   1:L PR[91] R[100]mm/sec CNT100;
   1:  PR[91,1] = PR[90,1] + 37.532;
   1:  PR[91,2] = PR[90,2] + 2.795;
   1:L PR[91] R[100]mm/sec CNT100;
   1:  PR[91,1] = PR[90,1] + 37.500;
   1:  PR[91,2] = PR[90,2] + 3.023;
   1:L PR[91] R[100]mm/sec CNT100;
   1:  PR[91,1] = PR[90,1] + 36.763;
   1:  PR[91,2] = PR[90,2] + 5.831;
   1:L PR[91] R[100]mm/sec CNT100;
   1:  PR[91,1] = PR[90,1] + 35.316;
   1:  PR[91,2] = PR[90,2] + 9.032;
   1:L PR[91] R[100]mm/sec CNT100;
   1:  PR[91,1] = PR[90,1] + 33.687;
   1:  PR[91,2] = PR[90,2] + 11.493;
   1:L PR[91] R[100]mm/sec CNT100;
   1:  PR[91,1] = PR[90,1] + 33.253;
   1:  PR[91,2] = PR[90,2] + 12.032;
   1:L PR[91] R[100]mm/sec CNT100;
   1:  PR[91,1] = PR[90,1] + 31.314;
   1:  PR[91,2] = PR[90,2] + 14.124;
   1:L PR[91] R[100]mm/sec CNT100;
   1:  PR[91,1] = PR[90,1] + 29.228;
   1:  PR[91,2] = PR[90,2] + 15.750;
   1:L PR[91] R[100]mm/sec CNT100;
   1:  PR[91,1] = PR[90,1] + 28.265;
   1:  PR[91,2] = PR[90,2] + 16.449;
   1:L PR[91] R[100]mm/sec CNT100;
   1:  PR[91,1] = PR[90,1] + 26.032;
   1:  PR[91,2] = PR[90,2] + 17.693;
   1:L PR[91] R[100]mm/sec CNT100;
   1:  PR[91,1] = PR[90,1] + 23.783;
   1:  PR[91,2] = PR[90,2] + 18.520;
   1:L PR[91] R[100]mm/sec CNT100;
   1:  PR[91,1] = PR[90,1] + 22.146;
   1:  PR[91,2] = PR[90,2] + 19.160;
   1:L PR[91] R[100]mm/sec CNT100;
   1:  PR[91,1] = PR[90,1] + 19.988;
   1:  PR[91,2] = PR[90,2] + 19.606;
   1:L PR[91] R[100]mm/sec CNT100;
   1:  PR[91,1] = PR[90,1] + 17.828;
   1:  PR[91,2] = PR[90,2] + 19.862;
   1:L PR[91] R[100]mm/sec CNT100;
   1:  PR[91,1] = PR[90,1] + 15.729;
   1:  PR[91,2] = PR[90,2] + 19.971;
   1:L PR[91] R[100]mm/sec CNT100;
   1:  PR[91,1] = PR[90,1] + 13.857;
   1:  PR[91,2] = PR[90,2] + 19.781;
   1:L PR[91] R[100]mm/sec CNT100;
   1:  PR[91,1] = PR[90,1] + 11.168;
   1:  PR[91,2] = PR[90,2] + 19.409;
   1:L PR[91] R[100]mm/sec CNT100;
   1:  PR[91,1] = PR[90,1] + 9.530;
   1:  PR[91,2] = PR[90,2] + 18.985;
   1:L PR[91] R[100]mm/sec CNT100;
   1:  PR[91,1] = PR[90,1] + 8.064;
   1:  PR[91,2] = PR[90,2] + 18.343;
   1:L PR[91] R[100]mm/sec CNT100;
   1:  PR[91,1] = PR[90,1] + 5.139;
   1:  PR[91,2] = PR[90,2] + 17.121;
   1:L PR[91] R[100]mm/sec CNT100;
   1:  PR[91,1] = PR[90,1] + 3.965;
   1:  PR[91,2] = PR[90,2] + 16.371;
   1:L PR[91] R[100]mm/sec CNT100;
   1:  PR[91,1] = PR[90,1] + 3.405;
   1:  PR[91,2] = PR[90,2] + 15.985;
   1:L PR[91] R[100]mm/sec CNT100;
   1:  PR[91,1] = PR[90,1] + 2.387;
   1:  PR[91,2] = PR[90,2] + 15.179;
   1:L PR[91] R[100]mm/sec CNT100;
   1:  PR[91,1] = PR[90,1] + 2.008;
   1:  PR[91,2] = PR[90,2] + 14.843;
   1:L PR[91] R[100]mm/sec CNT100;
   1:  PR[91,1] = PR[90,1] + 1.924;
   1:  PR[91,2] = PR[90,2] + 14.787;
   1:L PR[91] R[100]mm/sec CNT100;
   1:  PR[91,1] = PR[90,1] + 1.541;
   1:  PR[91,2] = PR[90,2] + 14.416;
   1:L PR[91] R[100]mm/sec CNT100;
   1:  PR[91,1] = PR[90,1] + 0.779;
   1:  PR[91,2] = PR[90,2] + 14.285;
   1:L PR[91] R[100]mm/sec CNT100;
   1:  PR[91,1] = PR[90,1] + 0.419;
   1:  PR[91,2] = PR[90,2] + 14.088;
   1:L PR[91] R[100]mm/sec CNT100;
   1:  PR[91,1] = PR[90,1] + -0.391;
   1:L PR[91] R[100]mm/sec CNT100;
   1:  PR[91] = PR[90];
   1:  PR[91,1] = PR[90,1] + -1.750;
   1:  PR[91,2] = PR[90,2] + 15.019;
   1:  PR[91,3] = PR[90,3] + 33.245;
   1:L PR[91] R[100]mm/sec CNT100;
   1:  PR[91,1] = PR[90,1] + -1.966;
   1:  PR[91,2] = PR[90,2] + 15.226;
   1:L PR[91] R[100]mm/sec CNT100;
   1:  PR[91,1] = PR[90,1] + -3.004;
   1:  PR[91,2] = PR[90,2] + 16.046;
   1:L PR[91] R[100]mm/sec CNT100;
   1:  PR[91,1] = PR[90,1] + -3.762;
   1:  PR[91,2] = PR[90,2] + 16.531;
   1:L PR[91] R[100]mm/sec CNT100;
   1:  PR[91,1] = PR[90,1] + -4.723;
   1:  PR[91,2] = PR[90,2] + 17.176;
   1:L PR[91] R[100]mm/sec CNT100;
   1:  PR[91,1] = PR[90,1] + -6.056;
   1:  PR[91,2] = PR[90,2] + 17.758;
   1:L PR[91] R[100]mm/sec CNT100;
   1:  PR[91,1] = PR[90,1] + -9.172;
   1:  PR[91,2] = PR[90,2] + 19.064;
   1:L PR[91] R[100]mm/sec CNT100;
   1:  PR[91,1] = PR[90,1] + -10.666;
   1:  PR[91,2] = PR[90,2] + 19.451;
   1:L PR[91] R[100]mm/sec CNT100;
   1:  PR[91,1] = PR[90,1] + -12.540;
   1:  PR[91,2] = PR[90,2] + 19.646;
   1:L PR[91] R[100]mm/sec CNT100;
   1:  PR[91,1] = PR[90,1] + -15.381;
   1:  PR[91,2] = PR[90,2] + 20.034;
   1:L PR[91] R[100]mm/sec CNT100;
   1:  PR[91,1] = PR[90,1] + -17.322;
   1:  PR[91,2] = PR[90,2] + 19.931;
   1:L PR[91] R[100]mm/sec CNT100;
   1:  PR[91,1] = PR[90,1] + -19.724;
   1:  PR[91,2] = PR[90,2] + 19.647;
   1:L PR[91] R[100]mm/sec CNT100;
   1:  PR[91,1] = PR[90,1] + -21.764;
   1:  PR[91,2] = PR[90,2] + 19.224;
   1:L PR[91] R[100]mm/sec CNT100;
   1:  PR[91,1] = PR[90,1] + -24.013;
   1:  PR[91,2] = PR[90,2] + 18.389;
   1:L PR[91] R[100]mm/sec CNT100;
   1:  PR[91,1] = PR[90,1] + -25.716;
   1:  PR[91,2] = PR[90,2] + 17.723;
   1:L PR[91] R[100]mm/sec CNT100;
   1:  PR[91,1] = PR[90,1] + -27.825;
   1:  PR[91,2] = PR[90,2] + 16.541;
   1:L PR[91] R[100]mm/sec CNT100;
   1:  PR[91,1] = PR[90,1] + -30.010;
   1:  PR[91,2] = PR[90,2] + 14.841;
   1:L PR[91] R[100]mm/sec CNT100;
   1:  PR[91,1] = PR[90,1] + -31.019;
   1:  PR[91,2] = PR[90,2] + 14.106;
   1:L PR[91] R[100]mm/sec CNT100;
   1:  PR[91,1] = PR[90,1] + -32.838;
   1:  PR[91,2] = PR[90,2] + 12.142;
   1:L PR[91] R[100]mm/sec CNT100;
   1:  PR[91,1] = PR[90,1] + -33.428;
   1:  PR[91,2] = PR[90,2] + 11.409;
   1:L PR[91] R[100]mm/sec CNT100;
   1:  PR[91,1] = PR[90,1] + -34.956;
   1:  PR[91,2] = PR[90,2] + 9.087;
   1:L PR[91] R[100]mm/sec CNT100;
   1:  PR[91,1] = PR[90,1] + -36.446;
   1:  PR[91,2] = PR[90,2] + 5.748;
   1:L PR[91] R[100]mm/sec CNT100;
   1:  PR[91,1] = PR[90,1] + -37.137;
   1:  PR[91,2] = PR[90,2] + 3.081;
   1:L PR[91] R[100]mm/sec CNT100;
   1:  PR[91,1] = PR[90,1] + -37.374;
   1:  PR[91,2] = PR[90,2] + 0.115;
   1:L PR[91] R[100]mm/sec CNT100;
   1:  PR[91,1] = PR[90,1] + -37.439;
   1:  PR[91,2] = PR[90,2] + -0.354;
   1:L PR[91] R[100]mm/sec CNT100;
   1:  PR[91,1] = PR[90,1] + -37.214;
   1:  PR[91,2] = PR[90,2] + -3.186;
   1:L PR[91] R[100]mm/sec CNT100;
   1:  PR[91,1] = PR[90,1] + -37.147;
   1:  PR[91,2] = PR[90,2] + -3.665;
   1:L PR[91] R[100]mm/sec CNT100;
   1:  PR[91,1] = PR[90,1] + -36.446;
   1:  PR[91,2] = PR[90,2] + -6.371;
   1:L PR[91] R[100]mm/sec CNT100;
   1:  PR[91,1] = PR[90,1] + -35.239;
   1:  PR[91,2] = PR[90,2] + -9.063;
   1:L PR[91] R[100]mm/sec CNT100;
   1:  PR[91,1] = PR[90,1] + -34.952;
   1:  PR[91,2] = PR[90,2] + -9.717;
   1:L PR[91] R[100]mm/sec CNT100;
   1:  PR[91,1] = PR[90,1] + -33.427;
   1:  PR[91,2] = PR[90,2] + -12.034;
   1:L PR[91] R[100]mm/sec CNT100;
   1:  PR[91,1] = PR[90,1] + -32.835;
   1:  PR[91,2] = PR[90,2] + -12.768;
   1:L PR[91] R[100]mm/sec CNT100;
   1:  PR[91,1] = PR[90,1] + -30.998;
   1:  PR[91,2] = PR[90,2] + -14.752;
   1:L PR[91] R[100]mm/sec CNT100;
   1:  PR[91,1] = PR[90,1] + -29.002;
   1:  PR[91,2] = PR[90,2] + -16.314;
   1:L PR[91] R[100]mm/sec CNT100;
   1:  PR[91,1] = PR[90,1] + -27.839;
   1:  PR[91,2] = PR[90,2] + -17.157;
   1:L PR[91] R[100]mm/sec CNT100;
   1:  PR[91,1] = PR[90,1] + -25.720;
   1:  PR[91,2] = PR[90,2] + -18.345;
   1:L PR[91] R[100]mm/sec CNT100;
   1:  PR[91,1] = PR[90,1] + -23.597;
   1:  PR[91,2] = PR[90,2] + -19.129;
   1:L PR[91] R[100]mm/sec CNT100;
   1:  PR[91,1] = PR[90,1] + -21.738;
   1:  PR[91,2] = PR[90,2] + -19.854;
   1:L PR[91] R[100]mm/sec CNT100;
   1:  PR[91,1] = PR[90,1] + -19.710;
   1:  PR[91,2] = PR[90,2] + -20.274;
   1:L PR[91] R[100]mm/sec CNT100;
   1:  PR[91,1] = PR[90,1] + -17.303;
   1:  PR[91,2] = PR[90,2] + -20.555;
   1:L PR[91] R[100]mm/sec CNT100;
   1:  PR[91,1] = PR[90,1] + -15.334;
   1:  PR[91,2] = PR[90,2] + -20.659;
   1:L PR[91] R[100]mm/sec CNT100;
   1:  PR[91,1] = PR[90,1] + -13.585;
   1:  PR[91,2] = PR[90,2] + -20.483;
   1:L PR[91] R[100]mm/sec CNT100;
   1:  PR[91,1] = PR[90,1] + -10.663;
   1:  PR[91,2] = PR[90,2] + -20.074;
   1:L PR[91] R[100]mm/sec CNT100;
   1:  PR[91,1] = PR[90,1] + -9.156;
   1:  PR[91,2] = PR[90,2] + -19.684;
   1:L PR[91] R[100]mm/sec CNT100;
   1:  PR[91,1] = PR[90,1] + -7.803;
   1:  PR[91,2] = PR[90,2] + -19.090;
   1:L PR[91] R[100]mm/sec CNT100;
   1:  PR[91,1] = PR[90,1] + -4.609;
   1:  PR[91,2] = PR[90,2] + -17.729;
   1:L PR[91] R[100]mm/sec CNT100;
   1:  PR[91,1] = PR[90,1] + -3.572;
   1:  PR[91,2] = PR[90,2] + -17.067;
   1:L PR[91] R[100]mm/sec CNT100;
   1:  PR[91,1] = PR[90,1] + -2.643;
   1:  PR[91,2] = PR[90,2] + -16.396;
   1:L PR[91] R[100]mm/sec CNT100;
   1:  PR[91,1] = PR[90,1] + -1.685;
   1:  PR[91,2] = PR[90,2] + -15.558;
   1:L PR[91] R[100]mm/sec CNT100;
   1:  PR[91,1] = PR[90,1] + -0.884;
   1:  PR[91,2] = PR[90,2] + -15.285;
   1:L PR[91] R[100]mm/sec CNT100;
   1:  PR[91,1] = PR[90,1] + -0.313;
   1:  PR[91,2] = PR[90,2] + -14.848;
   1:L PR[91] R[100]mm/sec CNT100;
   1:  PR[91,1] = PR[90,1] + 0.513;
   1:  PR[91,2] = PR[90,2] + -15.142;
   1:L PR[91] R[100]mm/sec CNT100;
   1:  PR[91,1] = PR[90,1] + 1.632;
   1:  PR[91,2] = PR[90,2] + -15.342;
   1:L PR[91] R[100]mm/sec CNT100;
   1:  PR[91,1] = PR[90,1] + 1.864;
   1:  PR[91,2] = PR[90,2] + -15.606;
   1:L PR[91] R[100]mm/sec CNT100;
   1:  PR[91,1] = PR[90,1] + 1.960;
   1:  PR[91,2] = PR[90,2] + -15.664;
   1:L PR[91] R[100]mm/sec CNT100;
   1:  PR[91,1] = PR[90,1] + 2.771;
   1:  PR[91,2] = PR[90,2] + -16.374;
   1:L PR[91] R[100]mm/sec CNT100;
   1:  PR[91,1] = PR[90,1] + 3.240;
   1:  PR[91,2] = PR[90,2] + -16.675;
   1:L PR[91] R[100]mm/sec CNT100;
   1:  PR[91,1] = PR[90,1] + 3.869;
   1:  PR[91,2] = PR[90,2] + -17.123;
   1:L PR[91] R[100]mm/sec CNT100;
   1:  PR[91,1] = PR[90,1] + 4.780;
   1:  PR[91,2] = PR[90,2] + -17.738;
   1:L PR[91] R[100]mm/sec CNT100;
   1:  PR[91,1] = PR[90,1] + 9.302;
   1:  PR[91,2] = PR[90,2] + -19.679;
   1:L PR[91] R[100]mm/sec CNT100;
   1:  PR[91,1] = PR[90,1] + 10.793;
   1:  PR[91,2] = PR[90,2] + -20.065;
   1:L PR[91] R[100]mm/sec CNT100;
   1:  PR[91,1] = PR[90,1] + 12.664;
   1:  PR[91,2] = PR[90,2] + -20.262;
   1:L PR[91] R[100]mm/sec CNT100;
   1:  PR[91,1] = PR[90,1] + 15.511;
   1:  PR[91,2] = PR[90,2] + -20.658;
   1:L PR[91] R[100]mm/sec CNT100;
   1:  PR[91,1] = PR[90,1] + 17.443;
   1:  PR[91,2] = PR[90,2] + -20.557;
   1:L PR[91] R[100]mm/sec CNT100;
   1:  PR[91,1] = PR[90,1] + 19.851;
   1:  PR[91,2] = PR[90,2] + -20.277;
   1:L PR[91] R[100]mm/sec CNT100;
   1:  PR[91,1] = PR[90,1] + 21.888;
   1:  PR[91,2] = PR[90,2] + -19.855;
   1:L PR[91] R[100]mm/sec CNT100;
   1:  PR[91,1] = PR[90,1] + 24.142;
   1:  PR[91,2] = PR[90,2] + -19.022;
   1:L PR[91] R[100]mm/sec CNT100;
   1:  PR[91,1] = PR[90,1] + 25.852;
   1:  PR[91,2] = PR[90,2] + -18.358;
   1:L PR[91] R[100]mm/sec CNT100;
   1:  PR[91,1] = PR[90,1] + 27.952;
   1:  PR[91,2] = PR[90,2] + -17.187;
   1:L PR[91] R[100]mm/sec CNT100;
   1:  PR[91,1] = PR[90,1] + 30.119;
   1:  PR[91,2] = PR[90,2] + -15.508;
   1:L PR[91] R[100]mm/sec CNT100;
   1:  PR[91,1] = PR[90,1] + 31.133;
   1:  PR[91,2] = PR[90,2] + -14.771;
   1:L PR[91] R[100]mm/sec CNT100;
   1:  PR[91,1] = PR[90,1] + 32.956;
   1:  PR[91,2] = PR[90,2] + -12.805;
   1:L PR[91] R[100]mm/sec CNT100;
   1:  PR[91,1] = PR[90,1] + 33.551;
   1:  PR[91,2] = PR[90,2] + -12.066;
   1:L PR[91] R[100]mm/sec CNT100;
   1:  PR[91,1] = PR[90,1] + 35.101;
   1:  PR[91,2] = PR[90,2] + -9.725;
   1:L PR[91] R[100]mm/sec CNT100;
   1:  PR[91,1] = PR[90,1] + 36.351;
   1:  PR[91,2] = PR[90,2] + -6.972;
   1:L PR[91] R[100]mm/sec CNT100;
   1:  PR[91,1] = PR[90,1] + 36.587;
   1:  PR[91,2] = PR[90,2] + -6.435;
   1:L PR[91] R[100]mm/sec CNT100;
   1:  PR[91,1] = PR[90,1] + 37.280;
   1:  PR[91,2] = PR[90,2] + -3.795;
   1:L PR[91] R[100]mm/sec CNT100;
   1:  PR[91,1] = PR[90,1] + 37.531;
   1:  PR[91,2] = PR[90,2] + -0.740;
   1:L PR[91] R[100]mm/sec CNT100;
   1:  PR[91,1] = PR[90,1] + 37.596;
   1:  PR[91,2] = PR[90,2] + -0.271;
   1:L PR[91] R[100]mm/sec CNT100;
   1:  PR[91,1] = PR[90,1] + 37.358;
   1:  PR[91,2] = PR[90,2] + 2.651;
   1:L PR[91] R[100]mm/sec CNT100;
   1:  PR[91,1] = PR[90,1] + 37.291;
   1:  PR[91,2] = PR[90,2] + 3.131;
   1:L PR[91] R[100]mm/sec CNT100;
   1:  PR[91,1] = PR[90,1] + 36.589;
   1:  PR[91,2] = PR[90,2] + 5.804;
   1:L PR[91] R[100]mm/sec CNT100;
   1:  PR[91,1] = PR[90,1] + 35.101;
   1:  PR[91,2] = PR[90,2] + 9.100;
   1:L PR[91] R[100]mm/sec CNT100;
   1:  PR[91,1] = PR[90,1] + 33.552;
   1:  PR[91,2] = PR[90,2] + 11.440;
   1:L PR[91] R[100]mm/sec CNT100;
   1:  PR[91,1] = PR[90,1] + 32.959;
   1:  PR[91,2] = PR[90,2] + 12.178;
   1:L PR[91] R[100]mm/sec CNT100;
   1:  PR[91,1] = PR[90,1] + 31.120;
   1:  PR[91,2] = PR[90,2] + 14.162;
   1:L PR[91] R[100]mm/sec CNT100;
   1:  PR[91,1] = PR[90,1] + 29.140;
   1:  PR[91,2] = PR[90,2] + 15.704;
   1:L PR[91] R[100]mm/sec CNT100;
   1:  PR[91,1] = PR[90,1] + 27.979;
   1:  PR[91,2] = PR[90,2] + 16.549;
   1:L PR[91] R[100]mm/sec CNT100;
   1:  PR[91,1] = PR[90,1] + 25.871;
   1:  PR[91,2] = PR[90,2] + 17.723;
   1:L PR[91] R[100]mm/sec CNT100;
   1:  PR[91,1] = PR[90,1] + 23.744;
   1:  PR[91,2] = PR[90,2] + 18.504;
   1:L PR[91] R[100]mm/sec CNT100;
   1:  PR[91,1] = PR[90,1] + 21.888;
   1:  PR[91,2] = PR[90,2] + 19.230;
   1:L PR[91] R[100]mm/sec CNT100;
   1:  PR[91,1] = PR[90,1] + 19.864;
   1:  PR[91,2] = PR[90,2] + 19.649;
   1:L PR[91] R[100]mm/sec CNT100;
   1:  PR[91,1] = PR[90,1] + 17.462;
   1:  PR[91,2] = PR[90,2] + 19.933;
   1:L PR[91] R[100]mm/sec CNT100;
   1:  PR[91,1] = PR[90,1] + 15.505;
   1:  PR[91,2] = PR[90,2] + 20.035;
   1:L PR[91] R[100]mm/sec CNT100;
   1:  PR[91,1] = PR[90,1] + 13.759;
   1:  PR[91,2] = PR[90,2] + 19.858;
   1:L PR[91] R[100]mm/sec CNT100;
   1:  PR[91,1] = PR[90,1] + 10.843;
   1:  PR[91,2] = PR[90,2] + 19.455;
   1:L PR[91] R[100]mm/sec CNT100;
   1:  PR[91,1] = PR[90,1] + 9.334;
   1:  PR[91,2] = PR[90,2] + 19.064;
   1:L PR[91] R[100]mm/sec CNT100;
   1:  PR[91,1] = PR[90,1] + 7.979;
   1:  PR[91,2] = PR[90,2] + 18.471;
   1:L PR[91] R[100]mm/sec CNT100;
   1:  PR[91,1] = PR[90,1] + 4.851;
   1:  PR[91,2] = PR[90,2] + 17.164;
   1:L PR[91] R[100]mm/sec CNT100;
   1:  PR[91,1] = PR[90,1] + 3.782;
   1:  PR[91,2] = PR[90,2] + 16.481;
   1:L PR[91] R[100]mm/sec CNT100;
   1:  PR[91,1] = PR[90,1] + 3.184;
   1:  PR[91,2] = PR[90,2] + 16.068;
   1:L PR[91] R[100]mm/sec CNT100;
   1:  PR[91,1] = PR[90,1] + 2.112;
   1:  PR[91,2] = PR[90,2] + 15.220;
   1:L PR[91] R[100]mm/sec CNT100;
   1:  PR[91,1] = PR[90,1] + 1.543;
   1:  PR[91,2] = PR[90,2] + 14.693;
   1:L PR[91] R[100]mm/sec CNT100;
   1:  PR[91,1] = PR[90,1] + 0.620;
   1:  PR[91,2] = PR[90,2] + 14.535;
   1:L PR[91] R[100]mm/sec CNT100;
   1:  PR[91,1] = PR[90,1] + 0.378;
   1:  PR[91,2] = PR[90,2] + 14.403;
   1:L PR[91] R[100]mm/sec CNT100;
   1:  PR[91,1] = PR[90,1] + -0.366;
   1:L PR[91] R[100]mm/sec CNT100;
   1:  PR[91] = PR[90];
   1:  PR[91,1] = PR[90,1] + -1.654;
   1:  PR[91,2] = PR[90,2] + 15.236;
   1:  PR[91,3] = PR[90,3] + 33.855;
   1:L PR[91] R[100]mm/sec CNT100;
   1:  PR[91,1] = PR[90,1] + -2.784;
   1:  PR[91,2] = PR[90,2] + 16.130;
   1:L PR[91] R[100]mm/sec CNT100;
   1:  PR[91,1] = PR[90,1] + -3.408;
   1:  PR[91,2] = PR[90,2] + 16.530;
   1:L PR[91] R[100]mm/sec CNT100;
   1:  PR[91,1] = PR[90,1] + -4.436;
   1:  PR[91,2] = PR[90,2] + 17.219;
   1:L PR[91] R[100]mm/sec CNT100;
   1:  PR[91,1] = PR[90,1] + -5.640;
   1:  PR[91,2] = PR[90,2] + 17.745;
   1:L PR[91] R[100]mm/sec CNT100;
   1:  PR[91,1] = PR[90,1] + -8.977;
   1:  PR[91,2] = PR[90,2] + 19.143;
   1:L PR[91] R[100]mm/sec CNT100;
   1:  PR[91,1] = PR[90,1] + -10.341;
   1:  PR[91,2] = PR[90,2] + 19.496;
   1:L PR[91] R[100]mm/sec CNT100;
   1:  PR[91,1] = PR[90,1] + -12.067;
   1:  PR[91,2] = PR[90,2] + 19.676;
   1:L PR[91] R[100]mm/sec CNT100;
   1:  PR[91,1] = PR[90,1] + -15.157;
   1:  PR[91,2] = PR[90,2] + 20.098;
   1:L PR[91] R[100]mm/sec CNT100;
   1:  PR[91,1] = PR[90,1] + -16.955;
   1:  PR[91,2] = PR[90,2] + 20.003;
   1:L PR[91] R[100]mm/sec CNT100;
   1:  PR[91,1] = PR[90,1] + -19.599;
   1:  PR[91,2] = PR[90,2] + 19.690;
   1:L PR[91] R[100]mm/sec CNT100;
   1:  PR[91,1] = PR[90,1] + -21.505;
   1:  PR[91,2] = PR[90,2] + 19.294;
   1:L PR[91] R[100]mm/sec CNT100;
   1:  PR[91,1] = PR[90,1] + -23.612;
   1:  PR[91,2] = PR[90,2] + 18.513;
   1:L PR[91] R[100]mm/sec CNT100;
   1:  PR[91,1] = PR[90,1] + -25.554;
   1:  PR[91,2] = PR[90,2] + 17.753;
   1:L PR[91] R[100]mm/sec CNT100;
   1:  PR[91,1] = PR[90,1] + -27.537;
   1:  PR[91,2] = PR[90,2] + 16.642;
   1:L PR[91] R[100]mm/sec CNT100;
   1:  PR[91,1] = PR[90,1] + -29.598;
   1:  PR[91,2] = PR[90,2] + 15.038;
   1:L PR[91] R[100]mm/sec CNT100;
   1:  PR[91,1] = PR[90,1] + -30.823;
   1:  PR[91,2] = PR[90,2] + 14.146;
   1:L PR[91] R[100]mm/sec CNT100;
   1:  PR[91,1] = PR[90,1] + -32.542;
   1:  PR[91,2] = PR[90,2] + 12.290;
   1:L PR[91] R[100]mm/sec CNT100;
   1:  PR[91,1] = PR[90,1] + -33.292;
   1:  PR[91,2] = PR[90,2] + 11.357;
   1:L PR[91] R[100]mm/sec CNT100;
   1:  PR[91,1] = PR[90,1] + -34.740;
   1:  PR[91,2] = PR[90,2] + 9.157;
   1:L PR[91] R[100]mm/sec CNT100;
   1:  PR[91,1] = PR[90,1] + -36.271;
   1:  PR[91,2] = PR[90,2] + 5.723;
   1:L PR[91] R[100]mm/sec CNT100;
   1:  PR[91,1] = PR[90,1] + -36.927;
   1:  PR[91,2] = PR[90,2] + 3.192;
   1:L PR[91] R[100]mm/sec CNT100;
   1:  PR[91,1] = PR[90,1] + -37.152;
   1:  PR[91,2] = PR[90,2] + 0.370;
   1:L PR[91] R[100]mm/sec CNT100;
   1:  PR[91,1] = PR[90,1] + -37.253;
   1:  PR[91,2] = PR[90,2] + -0.354;
   1:L PR[91] R[100]mm/sec CNT100;
   1:  PR[91,1] = PR[90,1] + -37.039;
   1:  PR[91,2] = PR[90,2] + -3.046;
   1:L PR[91] R[100]mm/sec CNT100;
   1:  PR[91,1] = PR[90,1] + -36.937;
   1:  PR[91,2] = PR[90,2] + -3.776;
   1:L PR[91] R[100]mm/sec CNT100;
   1:  PR[91,1] = PR[90,1] + -36.272;
   1:  PR[91,2] = PR[90,2] + -6.346;
   1:L PR[91] R[100]mm/sec CNT100;
   1:  PR[91,1] = PR[90,1] + -35.123;
   1:  PR[91,2] = PR[90,2] + -8.906;
   1:L PR[91] R[100]mm/sec CNT100;
   1:  PR[91,1] = PR[90,1] + -34.737;
   1:  PR[91,2] = PR[90,2] + -9.787;
   1:L PR[91] R[100]mm/sec CNT100;
   1:  PR[91,1] = PR[90,1] + -33.291;
   1:  PR[91,2] = PR[90,2] + -11.984;
   1:L PR[91] R[100]mm/sec CNT100;
   1:  PR[91,1] = PR[90,1] + -32.538;
   1:  PR[91,2] = PR[90,2] + -12.917;
   1:L PR[91] R[100]mm/sec CNT100;
   1:  PR[91,1] = PR[90,1] + -30.802;
   1:  PR[91,2] = PR[90,2] + -14.793;
   1:L PR[91] R[100]mm/sec CNT100;
   1:  PR[91,1] = PR[90,1] + -28.914;
   1:  PR[91,2] = PR[90,2] + -16.270;
   1:L PR[91] R[100]mm/sec CNT100;
   1:  PR[91,1] = PR[90,1] + -27.550;
   1:  PR[91,2] = PR[90,2] + -17.259;
   1:L PR[91] R[100]mm/sec CNT100;
   1:  PR[91,1] = PR[90,1] + -25.557;
   1:  PR[91,2] = PR[90,2] + -18.375;
   1:L PR[91] R[100]mm/sec CNT100;
   1:  PR[91,1] = PR[90,1] + -23.556;
   1:  PR[91,2] = PR[90,2] + -19.114;
   1:L PR[91] R[100]mm/sec CNT100;
   1:  PR[91,1] = PR[90,1] + -21.478;
   1:  PR[91,2] = PR[90,2] + -19.925;
   1:L PR[91] R[100]mm/sec CNT100;
   1:  PR[91,1] = PR[90,1] + -19.584;
   1:  PR[91,2] = PR[90,2] + -20.318;
   1:L PR[91] R[100]mm/sec CNT100;
   1:  PR[91,1] = PR[90,1] + -16.934;
   1:  PR[91,2] = PR[90,2] + -20.626;
   1:L PR[91] R[100]mm/sec CNT100;
   1:  PR[91,1] = PR[90,1] + -15.108;
   1:  PR[91,2] = PR[90,2] + -20.723;
   1:L PR[91] R[100]mm/sec CNT100;
   1:  PR[91,1] = PR[90,1] + -13.486;
   1:  PR[91,2] = PR[90,2] + -20.559;
   1:L PR[91] R[100]mm/sec CNT100;
   1:  PR[91,1] = PR[90,1] + -10.336;
   1:  PR[91,2] = PR[90,2] + -20.119;
   1:L PR[91] R[100]mm/sec CNT100;
   1:  PR[91,1] = PR[90,1] + -8.958;
   1:  PR[91,2] = PR[90,2] + -19.762;
   1:L PR[91] R[100]mm/sec CNT100;
   1:  PR[91,1] = PR[90,1] + -7.715;
   1:  PR[91,2] = PR[90,2] + -19.217;
   1:L PR[91] R[100]mm/sec CNT100;
   1:  PR[91,1] = PR[90,1] + -4.316;
   1:  PR[91,2] = PR[90,2] + -17.769;
   1:L PR[91] R[100]mm/sec CNT100;
   1:  PR[91,1] = PR[90,1] + -3.388;
   1:  PR[91,2] = PR[90,2] + -17.175;
   1:L PR[91] R[100]mm/sec CNT100;
   1:  PR[91,1] = PR[90,1] + -2.398;
   1:  PR[91,2] = PR[90,2] + -16.462;
   1:L PR[91] R[100]mm/sec CNT100;
   1:  PR[91,1] = PR[90,1] + -1.670;
   1:  PR[91,2] = PR[90,2] + -15.824;
   1:L PR[91] R[100]mm/sec CNT100;
   1:  PR[91,1] = PR[90,1] + -0.149;
   1:  PR[91,2] = PR[90,2] + -15.297;
   1:L PR[91] R[100]mm/sec CNT100;
   1:  PR[91,1] = PR[90,1] + 1.655;
   1:  PR[91,2] = PR[90,2] + -15.626;
   1:L PR[91] R[100]mm/sec CNT100;
   1:  PR[91,1] = PR[90,1] + 1.896;
   1:  PR[91,2] = PR[90,2] + -15.900;
   1:L PR[91] R[100]mm/sec CNT100;
   1:  PR[91,1] = PR[90,1] + 1.942;
   1:  PR[91,2] = PR[90,2] + -15.927;
   1:L PR[91] R[100]mm/sec CNT100;
   1:  PR[91,1] = PR[90,1] + 2.525;
   1:  PR[91,2] = PR[90,2] + -16.439;
   1:L PR[91] R[100]mm/sec CNT100;
   1:  PR[91,1] = PR[90,1] + 2.844;
   1:  PR[91,2] = PR[90,2] + -16.643;
   1:L PR[91] R[100]mm/sec CNT100;
   1:  PR[91,1] = PR[90,1] + 3.511;
   1:  PR[91,2] = PR[90,2] + -17.118;
   1:L PR[91] R[100]mm/sec CNT100;
   1:  PR[91,1] = PR[90,1] + 4.486;
   1:  PR[91,2] = PR[90,2] + -17.777;
   1:L PR[91] R[100]mm/sec CNT100;
   1:  PR[91,1] = PR[90,1] + 9.104;
   1:  PR[91,2] = PR[90,2] + -19.757;
   1:L PR[91] R[100]mm/sec CNT100;
   1:  PR[91,1] = PR[90,1] + 10.466;
   1:  PR[91,2] = PR[90,2] + -20.110;
   1:L PR[91] R[100]mm/sec CNT100;
   1:  PR[91,1] = PR[90,1] + 12.188;
   1:  PR[91,2] = PR[90,2] + -20.291;
   1:L PR[91] R[100]mm/sec CNT100;
   1:  PR[91,1] = PR[90,1] + 15.286;
   1:  PR[91,2] = PR[90,2] + -20.722;
   1:L PR[91] R[100]mm/sec CNT100;
   1:  PR[91,1] = PR[90,1] + 17.075;
   1:  PR[91,2] = PR[90,2] + -20.629;
   1:L PR[91] R[100]mm/sec CNT100;
   1:  PR[91,1] = PR[90,1] + 19.726;
   1:  PR[91,2] = PR[90,2] + -20.320;
   1:L PR[91] R[100]mm/sec CNT100;
   1:  PR[91,1] = PR[90,1] + 21.629;
   1:  PR[91,2] = PR[90,2] + -19.926;
   1:L PR[91] R[100]mm/sec CNT100;
   1:  PR[91,1] = PR[90,1] + 23.740;
   1:  PR[91,2] = PR[90,2] + -19.146;
   1:L PR[91] R[100]mm/sec CNT100;
   1:  PR[91,1] = PR[90,1] + 25.690;
   1:  PR[91,2] = PR[90,2] + -18.388;
   1:L PR[91] R[100]mm/sec CNT100;
   1:  PR[91,1] = PR[90,1] + 27.664;
   1:  PR[91,2] = PR[90,2] + -17.288;
   1:L PR[91] R[100]mm/sec CNT100;
   1:  PR[91,1] = PR[90,1] + 29.708;
   1:  PR[91,2] = PR[90,2] + -15.704;
   1:L PR[91] R[100]mm/sec CNT100;
   1:  PR[91,1] = PR[90,1] + 30.938;
   1:  PR[91,2] = PR[90,2] + -14.810;
   1:L PR[91] R[100]mm/sec CNT100;
   1:  PR[91,1] = PR[90,1] + 32.661;
   1:  PR[91,2] = PR[90,2] + -12.952;
   1:L PR[91] R[100]mm/sec CNT100;
   1:  PR[91,1] = PR[90,1] + 33.417;
   1:  PR[91,2] = PR[90,2] + -12.013;
   1:L PR[91] R[100]mm/sec CNT100;
   1:  PR[91,1] = PR[90,1] + 34.886;
   1:  PR[91,2] = PR[90,2] + -9.794;
   1:L PR[91] R[100]mm/sec CNT100;
   1:  PR[91,1] = PR[90,1] + 36.073;
   1:  PR[91,2] = PR[90,2] + -7.179;
   1:L PR[91] R[100]mm/sec CNT100;
   1:  PR[91,1] = PR[90,1] + 36.413;
   1:  PR[91,2] = PR[90,2] + -6.408;
   1:L PR[91] R[100]mm/sec CNT100;
   1:  PR[91,1] = PR[90,1] + 37.071;
   1:  PR[91,2] = PR[90,2] + -3.903;
   1:L PR[91] R[100]mm/sec CNT100;
   1:  PR[91,1] = PR[90,1] + 37.309;
   1:  PR[91,2] = PR[90,2] + -0.996;
   1:L PR[91] R[100]mm/sec CNT100;
   1:  PR[91,1] = PR[90,1] + 37.409;
   1:  PR[91,2] = PR[90,2] + -0.271;
   1:L PR[91] R[100]mm/sec CNT100;
   1:  PR[91,1] = PR[90,1] + 37.183;
   1:  PR[91,2] = PR[90,2] + 2.507;
   1:L PR[91] R[100]mm/sec CNT100;
   1:  PR[91,1] = PR[90,1] + 37.081;
   1:  PR[91,2] = PR[90,2] + 3.239;
   1:L PR[91] R[100]mm/sec CNT100;
   1:  PR[91,1] = PR[90,1] + 36.415;
   1:  PR[91,2] = PR[90,2] + 5.777;
   1:L PR[91] R[100]mm/sec CNT100;
   1:  PR[91,1] = PR[90,1] + 34.887;
   1:  PR[91,2] = PR[90,2] + 9.169;
   1:L PR[91] R[100]mm/sec CNT100;
   1:  PR[91,1] = PR[90,1] + 33.418;
   1:  PR[91,2] = PR[90,2] + 11.387;
   1:L PR[91] R[100]mm/sec CNT100;
   1:  PR[91,1] = PR[90,1] + 32.665;
   1:  PR[91,2] = PR[90,2] + 12.325;
   1:L PR[91] R[100]mm/sec CNT100;
   1:  PR[91,1] = PR[90,1] + 30.926;
   1:  PR[91,2] = PR[90,2] + 14.200;
   1:L PR[91] R[100]mm/sec CNT100;
   1:  PR[91,1] = PR[90,1] + 29.053;
   1:  PR[91,2] = PR[90,2] + 15.659;
   1:L PR[91] R[100]mm/sec CNT100;
   1:  PR[91,1] = PR[90,1] + 27.692;
   1:  PR[91,2] = PR[90,2] + 16.648;
   1:L PR[91] R[100]mm/sec CNT100;
   1:  PR[91,1] = PR[90,1] + 25.711;
   1:  PR[91,2] = PR[90,2] + 17.752;
   1:L PR[91] R[100]mm/sec CNT100;
   1:  PR[91,1] = PR[90,1] + 23.706;
   1:  PR[91,2] = PR[90,2] + 18.489;
   1:L PR[91] R[100]mm/sec CNT100;
   1:  PR[91,1] = PR[90,1] + 21.631;
   1:  PR[91,2] = PR[90,2] + 19.301;
   1:L PR[91] R[100]mm/sec CNT100;
   1:  PR[91,1] = PR[90,1] + 19.740;
   1:  PR[91,2] = PR[90,2] + 19.692;
   1:L PR[91] R[100]mm/sec CNT100;
   1:  PR[91,1] = PR[90,1] + 17.096;
   1:  PR[91,2] = PR[90,2] + 20.005;
   1:L PR[91] R[100]mm/sec CNT100;
   1:  PR[91,1] = PR[90,1] + 15.281;
   1:  PR[91,2] = PR[90,2] + 20.099;
   1:L PR[91] R[100]mm/sec CNT100;
   1:  PR[91,1] = PR[90,1] + 13.662;
   1:  PR[91,2] = PR[90,2] + 19.935;
   1:L PR[91] R[100]mm/sec CNT100;
   1:  PR[91,1] = PR[90,1] + 10.518;
   1:  PR[91,2] = PR[90,2] + 19.500;
   1:L PR[91] R[100]mm/sec CNT100;
   1:  PR[91,1] = PR[90,1] + 9.138;
   1:  PR[91,2] = PR[90,2] + 19.142;
   1:L PR[91] R[100]mm/sec CNT100;
   1:  PR[91,1] = PR[90,1] + 7.893;
   1:  PR[91,2] = PR[90,2] + 18.598;
   1:L PR[91] R[100]mm/sec CNT100;
   1:  PR[91,1] = PR[90,1] + 4.564;
   1:  PR[91,2] = PR[90,2] + 17.206;
   1:L PR[91] R[100]mm/sec CNT100;
   1:  PR[91,1] = PR[90,1] + 3.599;
   1:  PR[91,2] = PR[90,2] + 16.590;
   1:L PR[91] R[100]mm/sec CNT100;
   1:  PR[91,1] = PR[90,1] + 2.963;
   1:  PR[91,2] = PR[90,2] + 16.151;
   1:L PR[91] R[100]mm/sec CNT100;
   1:  PR[91,1] = PR[90,1] + 2.037;
   1:  PR[91,2] = PR[90,2] + 15.418;
   1:L PR[91] R[100]mm/sec CNT100;
   1:  PR[91,1] = PR[90,1] + 1.582;
   1:  PR[91,2] = PR[90,2] + 14.977;
   1:L PR[91] R[100]mm/sec CNT100;
   1:  PR[91,1] = PR[90,1] + -0.181;
   1:  PR[91,2] = PR[90,2] + 14.671;
   1:L PR[91] R[100]mm/sec CNT100;
   1:  PR[91] = PR[90];
   1:  PR[91,1] = PR[90,1] + -1.636;
   1:  PR[91,2] = PR[90,2] + 15.480;
   1:  PR[91,3] = PR[90,3] + 34.465;
   1:L PR[91] R[100]mm/sec CNT100;
   1:  PR[91,1] = PR[90,1] + -2.573;
   1:  PR[91,2] = PR[90,2] + 16.221;
   1:L PR[91] R[100]mm/sec CNT100;
   1:  PR[91,1] = PR[90,1] + -4.144;
   1:  PR[91,2] = PR[90,2] + 17.260;
   1:L PR[91] R[100]mm/sec CNT100;
   1:  PR[91,1] = PR[90,1] + -5.225;
   1:  PR[91,2] = PR[90,2] + 17.732;
   1:L PR[91] R[100]mm/sec CNT100;
   1:  PR[91,1] = PR[90,1] + -8.781;
   1:  PR[91,2] = PR[90,2] + 19.222;
   1:L PR[91] R[100]mm/sec CNT100;
   1:  PR[91,1] = PR[90,1] + -10.016;
   1:  PR[91,2] = PR[90,2] + 19.542;
   1:L PR[91] R[100]mm/sec CNT100;
   1:  PR[91,1] = PR[90,1] + -11.593;
   1:  PR[91,2] = PR[90,2] + 19.706;
   1:L PR[91] R[100]mm/sec CNT100;
   1:  PR[91,1] = PR[90,1] + -14.933;
   1:  PR[91,2] = PR[90,2] + 20.162;
   1:L PR[91] R[100]mm/sec CNT100;
   1:  PR[91,1] = PR[90,1] + -16.588;
   1:  PR[91,2] = PR[90,2] + 20.074;
   1:L PR[91] R[100]mm/sec CNT100;
   1:  PR[91,1] = PR[90,1] + -19.474;
   1:  PR[91,2] = PR[90,2] + 19.733;
   1:L PR[91] R[100]mm/sec CNT100;
   1:  PR[91,1] = PR[90,1] + -21.247;
   1:  PR[91,2] = PR[90,2] + 19.365;
   1:L PR[91] R[100]mm/sec CNT100;
   1:  PR[91,1] = PR[90,1] + -23.211;
   1:  PR[91,2] = PR[90,2] + 18.636;
   1:L PR[91] R[100]mm/sec CNT100;
   1:  PR[91,1] = PR[90,1] + -25.393;
   1:  PR[91,2] = PR[90,2] + 17.783;
   1:L PR[91] R[100]mm/sec CNT100;
   1:  PR[91,1] = PR[90,1] + -27.250;
   1:  PR[91,2] = PR[90,2] + 16.743;
   1:L PR[91] R[100]mm/sec CNT100;
   1:  PR[91,1] = PR[90,1] + -29.186;
   1:  PR[91,2] = PR[90,2] + 15.236;
   1:L PR[91] R[100]mm/sec CNT100;
   1:  PR[91,1] = PR[90,1] + -30.627;
   1:  PR[91,2] = PR[90,2] + 14.187;
   1:L PR[91] R[100]mm/sec CNT100;
   1:  PR[91,1] = PR[90,1] + -32.246;
   1:  PR[91,2] = PR[90,2] + 12.438;
   1:L PR[91] R[100]mm/sec CNT100;
   1:  PR[91,1] = PR[90,1] + -33.157;
   1:  PR[91,2] = PR[90,2] + 11.306;
   1:L PR[91] R[100]mm/sec CNT100;
   1:  PR[91,1] = PR[90,1] + -34.525;
   1:  PR[91,2] = PR[90,2] + 9.226;
   1:L PR[91] R[100]mm/sec CNT100;
   1:  PR[91,1] = PR[90,1] + -36.097;
   1:  PR[91,2] = PR[90,2] + 5.698;
   1:L PR[91] R[100]mm/sec CNT100;
   1:  PR[91,1] = PR[90,1] + -36.716;
   1:  PR[91,2] = PR[90,2] + 3.304;
   1:L PR[91] R[100]mm/sec CNT100;
   1:  PR[91,1] = PR[90,1] + -36.931;
   1:  PR[91,2] = PR[90,2] + 0.625;
   1:L PR[91] R[100]mm/sec CNT100;
   1:  PR[91,1] = PR[90,1] + -37.067;
   1:  PR[91,2] = PR[90,2] + -0.354;
   1:L PR[91] R[100]mm/sec CNT100;
   1:  PR[91,1] = PR[90,1] + -36.864;
   1:  PR[91,2] = PR[90,2] + -2.907;
   1:L PR[91] R[100]mm/sec CNT100;
   1:  PR[91,1] = PR[90,1] + -36.727;
   1:  PR[91,2] = PR[90,2] + -3.888;
   1:L PR[91] R[100]mm/sec CNT100;
   1:  PR[91,1] = PR[90,1] + -36.097;
   1:  PR[91,2] = PR[90,2] + -6.321;
   1:L PR[91] R[100]mm/sec CNT100;
   1:  PR[91,1] = PR[90,1] + -35.007;
   1:  PR[91,2] = PR[90,2] + -8.749;
   1:L PR[91] R[100]mm/sec CNT100;
   1:  PR[91,1] = PR[90,1] + -34.521;
   1:  PR[91,2] = PR[90,2] + -9.857;
   1:L PR[91] R[100]mm/sec CNT100;
   1:  PR[91,1] = PR[90,1] + -33.155;
   1:  PR[91,2] = PR[90,2] + -11.933;
   1:L PR[91] R[100]mm/sec CNT100;
   1:  PR[91,1] = PR[90,1] + -32.242;
   1:  PR[91,2] = PR[90,2] + -13.065;
   1:L PR[91] R[100]mm/sec CNT100;
   1:  PR[91,1] = PR[90,1] + -30.605;
   1:  PR[91,2] = PR[90,2] + -14.834;
   1:L PR[91] R[100]mm/sec CNT100;
   1:  PR[91,1] = PR[90,1] + -28.825;
   1:  PR[91,2] = PR[90,2] + -16.227;
   1:L PR[91] R[100]mm/sec CNT100;
   1:  PR[91,1] = PR[90,1] + -27.261;
   1:  PR[91,2] = PR[90,2] + -17.360;
   1:L PR[91] R[100]mm/sec CNT100;
   1:  PR[91,1] = PR[90,1] + -25.395;
   1:  PR[91,2] = PR[90,2] + -18.406;
   1:L PR[91] R[100]mm/sec CNT100;
   1:  PR[91,1] = PR[90,1] + -23.516;
   1:  PR[91,2] = PR[90,2] + -19.100;
   1:L PR[91] R[100]mm/sec CNT100;
   1:  PR[91,1] = PR[90,1] + -21.218;
   1:  PR[91,2] = PR[90,2] + -19.996;
   1:L PR[91] R[100]mm/sec CNT100;
   1:  PR[91,1] = PR[90,1] + -19.458;
   1:  PR[91,2] = PR[90,2] + -20.361;
   1:L PR[91] R[100]mm/sec CNT100;
   1:  PR[91,1] = PR[90,1] + -16.565;
   1:  PR[91,2] = PR[90,2] + -20.698;
   1:L PR[91] R[100]mm/sec CNT100;
   1:  PR[91,1] = PR[90,1] + -14.882;
   1:  PR[91,2] = PR[90,2] + -20.787;
   1:L PR[91] R[100]mm/sec CNT100;
   1:  PR[91,1] = PR[90,1] + -13.387;
   1:  PR[91,2] = PR[90,2] + -20.636;
   1:L PR[91] R[100]mm/sec CNT100;
   1:  PR[91,1] = PR[90,1] + -10.009;
   1:  PR[91,2] = PR[90,2] + -20.163;
   1:L PR[91] R[100]mm/sec CNT100;
   1:  PR[91,1] = PR[90,1] + -8.760;
   1:  PR[91,2] = PR[90,2] + -19.840;
   1:L PR[91] R[100]mm/sec CNT100;
   1:  PR[91,1] = PR[90,1] + -7.628;
   1:  PR[91,2] = PR[90,2] + -19.344;
   1:L PR[91] R[100]mm/sec CNT100;
   1:  PR[91,1] = PR[90,1] + -4.022;
   1:  PR[91,2] = PR[90,2] + -17.808;
   1:L PR[91] R[100]mm/sec CNT100;
   1:  PR[91,1] = PR[90,1] + -3.202;
   1:  PR[91,2] = PR[90,2] + -17.283;
   1:L PR[91] R[100]mm/sec CNT100;
   1:  PR[91,1] = PR[90,1] + -2.154;
   1:  PR[91,2] = PR[90,2] + -16.528;
   1:L PR[91] R[100]mm/sec CNT100;
   1:  PR[91,1] = PR[90,1] + -1.649;
   1:  PR[91,2] = PR[90,2] + -16.085;
   1:L PR[91] R[100]mm/sec CNT100;
   1:  PR[91,1] = PR[90,1] + -0.861;
   1:  PR[91,2] = PR[90,2] + -15.817;
   1:L PR[91] R[100]mm/sec CNT100;
   1:  PR[91,1] = PR[90,1] + -0.023;
   1:  PR[91,2] = PR[90,2] + -15.471;
   1:L PR[91] R[100]mm/sec CNT100;
   1:  PR[91,1] = PR[90,1] + 0.569;
   1:  PR[91,2] = PR[90,2] + -15.707;
   1:L PR[91] R[100]mm/sec CNT100;
   1:  PR[91,1] = PR[90,1] + 1.674;
   1:  PR[91,2] = PR[90,2] + -15.905;
   1:L PR[91] R[100]mm/sec CNT100;
   1:  PR[91,1] = PR[90,1] + 1.933;
   1:  PR[91,2] = PR[90,2] + -16.199;
   1:L PR[91] R[100]mm/sec CNT100;
   1:  PR[91,1] = PR[90,1] + 2.296;
   1:  PR[91,2] = PR[90,2] + -16.518;
   1:L PR[91] R[100]mm/sec CNT100;
   1:  PR[91,1] = PR[90,1] + 4.197;
   1:  PR[91,2] = PR[90,2] + -17.817;
   1:L PR[91] R[100]mm/sec CNT100;
   1:  PR[91,1] = PR[90,1] + 8.906;
   1:  PR[91,2] = PR[90,2] + -19.835;
   1:L PR[91] R[100]mm/sec CNT100;
   1:  PR[91,1] = PR[90,1] + 10.139;
   1:  PR[91,2] = PR[90,2] + -20.155;
   1:L PR[91] R[100]mm/sec CNT100;
   1:  PR[91,1] = PR[90,1] + 11.713;
   1:  PR[91,2] = PR[90,2] + -20.320;
   1:L PR[91] R[100]mm/sec CNT100;
   1:  PR[91,1] = PR[90,1] + 15.060;
   1:  PR[91,2] = PR[90,2] + -20.786;
   1:L PR[91] R[100]mm/sec CNT100;
   1:  PR[91,1] = PR[90,1] + 16.707;
   1:  PR[91,2] = PR[90,2] + -20.700;
   1:L PR[91] R[100]mm/sec CNT100;
   1:  PR[91,1] = PR[90,1] + 19.600;
   1:  PR[91,2] = PR[90,2] + -20.363;
   1:L PR[91] R[100]mm/sec CNT100;
   1:  PR[91,1] = PR[90,1] + 21.371;
   1:  PR[91,2] = PR[90,2] + -19.996;
   1:L PR[91] R[100]mm/sec CNT100;
   1:  PR[91,1] = PR[90,1] + 23.338;
   1:  PR[91,2] = PR[90,2] + -19.270;
   1:L PR[91] R[100]mm/sec CNT100;
   1:  PR[91,1] = PR[90,1] + 25.528;
   1:  PR[91,2] = PR[90,2] + -18.418;
   1:L PR[91] R[100]mm/sec CNT100;
   1:  PR[91,1] = PR[90,1] + 27.377;
   1:  PR[91,2] = PR[90,2] + -17.388;
   1:L PR[91] R[100]mm/sec CNT100;
   1:  PR[91,1] = PR[90,1] + 29.297;
   1:  PR[91,2] = PR[90,2] + -15.900;
   1:L PR[91] R[100]mm/sec CNT100;
   1:  PR[91,1] = PR[90,1] + 30.743;
   1:  PR[91,2] = PR[90,2] + -14.849;
   1:L PR[91] R[100]mm/sec CNT100;
   1:  PR[91,1] = PR[90,1] + 32.366;
   1:  PR[91,2] = PR[90,2] + -13.099;
   1:L PR[91] R[100]mm/sec CNT100;
   1:  PR[91,1] = PR[90,1] + 33.283;
   1:  PR[91,2] = PR[90,2] + -11.961;
   1:L PR[91] R[100]mm/sec CNT100;
   1:  PR[91,1] = PR[90,1] + 34.672;
   1:  PR[91,2] = PR[90,2] + -9.862;
   1:L PR[91] R[100]mm/sec CNT100;
   1:  PR[91,1] = PR[90,1] + 35.795;
   1:  PR[91,2] = PR[90,2] + -7.387;
   1:L PR[91] R[100]mm/sec CNT100;
   1:  PR[91,1] = PR[90,1] + 36.239;
   1:  PR[91,2] = PR[90,2] + -6.381;
   1:L PR[91] R[100]mm/sec CNT100;
   1:  PR[91,1] = PR[90,1] + 36.861;
   1:  PR[91,2] = PR[90,2] + -4.011;
   1:L PR[91] R[100]mm/sec CNT100;
   1:  PR[91,1] = PR[90,1] + 37.087;
   1:  PR[91,2] = PR[90,2] + -1.252;
   1:L PR[91] R[100]mm/sec CNT100;
   1:  PR[91,1] = PR[90,1] + 37.223;
   1:  PR[91,2] = PR[90,2] + -0.271;
   1:L PR[91] R[100]mm/sec CNT100;
   1:  PR[91,1] = PR[90,1] + 37.008;
   1:  PR[91,2] = PR[90,2] + 2.364;
   1:L PR[91] R[100]mm/sec CNT100;
   1:  PR[91,1] = PR[90,1] + 36.872;
   1:  PR[91,2] = PR[90,2] + 3.347;
   1:L PR[91] R[100]mm/sec CNT100;
   1:  PR[91,1] = PR[90,1] + 36.242;
   1:  PR[91,2] = PR[90,2] + 5.747;
   1:L PR[91] R[100]mm/sec CNT100;
   1:  PR[91,1] = PR[90,1] + 35.154;
   1:  PR[91,2] = PR[90,2] + 8.139;
   1:L PR[91] R[100]mm/sec CNT100;
   1:  PR[91,1] = PR[90,1] + 34.669;
   1:  PR[91,2] = PR[90,2] + 9.242;
   1:L PR[91] R[100]mm/sec CNT100;
   1:  PR[91,1] = PR[90,1] + 33.284;
   1:  PR[91,2] = PR[90,2] + 11.334;
   1:L PR[91] R[100]mm/sec CNT100;
   1:  PR[91,1] = PR[90,1] + 32.371;
   1:  PR[91,2] = PR[90,2] + 12.471;
   1:L PR[91] R[100]mm/sec CNT100;
   1:  PR[91,1] = PR[90,1] + 30.732;
   1:  PR[91,2] = PR[90,2] + 14.239;
   1:L PR[91] R[100]mm/sec CNT100;
   1:  PR[91,1] = PR[90,1] + 28.966;
   1:  PR[91,2] = PR[90,2] + 15.614;
   1:L PR[91] R[100]mm/sec CNT100;
   1:  PR[91,1] = PR[90,1] + 27.406;
   1:  PR[91,2] = PR[90,2] + 16.748;
   1:L PR[91] R[100]mm/sec CNT100;
   1:  PR[91,1] = PR[90,1] + 25.550;
   1:  PR[91,2] = PR[90,2] + 17.782;
   1:L PR[91] R[100]mm/sec CNT100;
   1:  PR[91,1] = PR[90,1] + 23.667;
   1:  PR[91,2] = PR[90,2] + 18.474;
   1:L PR[91] R[100]mm/sec CNT100;
   1:  PR[91,1] = PR[90,1] + 21.374;
   1:  PR[91,2] = PR[90,2] + 19.371;
   1:L PR[91] R[100]mm/sec CNT100;
   1:  PR[91,1] = PR[90,1] + 19.616;
   1:  PR[91,2] = PR[90,2] + 19.735;
   1:L PR[91] R[100]mm/sec CNT100;
   1:  PR[91,1] = PR[90,1] + 16.730;
   1:  PR[91,2] = PR[90,2] + 20.076;
   1:L PR[91] R[100]mm/sec CNT100;
   1:  PR[91,1] = PR[90,1] + 15.057;
   1:  PR[91,2] = PR[90,2] + 20.163;
   1:L PR[91] R[100]mm/sec CNT100;
   1:  PR[91,1] = PR[90,1] + 13.565;
   1:  PR[91,2] = PR[90,2] + 20.012;
   1:L PR[91] R[100]mm/sec CNT100;
   1:  PR[91,1] = PR[90,1] + 10.193;
   1:  PR[91,2] = PR[90,2] + 19.546;
   1:L PR[91] R[100]mm/sec CNT100;
   1:  PR[91,1] = PR[90,1] + 8.943;
   1:  PR[91,2] = PR[90,2] + 19.221;
   1:L PR[91] R[100]mm/sec CNT100;
   1:  PR[91,1] = PR[90,1] + 7.808;
   1:  PR[91,2] = PR[90,2] + 18.725;
   1:L PR[91] R[100]mm/sec CNT100;
   1:  PR[91,1] = PR[90,1] + 4.277;
   1:  PR[91,2] = PR[90,2] + 17.249;
   1:L PR[91] R[100]mm/sec CNT100;
   1:  PR[91,1] = PR[90,1] + 3.417;
   1:  PR[91,2] = PR[90,2] + 16.700;
   1:L PR[91] R[100]mm/sec CNT100;
   1:  PR[91,1] = PR[90,1] + 2.742;
   1:  PR[91,2] = PR[90,2] + 16.234;
   1:L PR[91] R[100]mm/sec CNT100;
   1:  PR[91,1] = PR[90,1] + 2.019;
   1:  PR[91,2] = PR[90,2] + 15.662;
   1:L PR[91] R[100]mm/sec CNT100;
   1:  PR[91,1] = PR[90,1] + 1.599;
   1:  PR[91,2] = PR[90,2] + 15.256;
   1:L PR[91] R[100]mm/sec CNT100;
   1:  PR[91,1] = PR[90,1] + 0.552;
   1:  PR[91,2] = PR[90,2] + 15.077;
   1:L PR[91] R[100]mm/sec CNT100;
   1:  PR[91,1] = PR[90,1] + -0.002;
   1:  PR[91,2] = PR[90,2] + 14.853;
   1:L PR[91] R[100]mm/sec CNT100 TB   .50sec,CALL END_PUD;
   1:  DO[117:Laser Start]=OFF;
   1:  PR[92] = PR[91];
   1:  PR[92,3] = PR[92,3] + 50;
   1:J PR[92] 10% FINE;
   1:  WAIT   5.00(sec);
   1:  DO[119:Gas]=OFF;
   1:  CALL HOME_ALL;
/POS
/END
